(* IEC 61131-3 sources: eCockpitGit/test_project/src/%F%00 Library/%F%Common Functions/%F%Bits/%F%Bit Get, 3 files *)

(* ---- %POU%FU_bBitGet.st ---- *)
//This function get the bit value from a variable
// |**Version**|**Author**| **Date** |**Changes**
// | 1         | NSN      | 11-01-19 | Creation
FUNCTION FU_bBitGet : BOOL
VAR_INPUT
	bVar	:BYTE;		//The value to work with
	bIndex	:BYTE;		//Which bit to get
END_VAR
(*%!%__DELIMITER__%!%*)
FU_bBitGet			:=		(bVar AND SHL(1,bIndex)) <> 0;

(* ---- %POU%FU_dwBitGet.st ---- *)
//This function get the bit value from a variable
// |**Version**|**Author**| **Date** |**Changes**
// | 1         | NSN      | 11-01-19 | Creation
FUNCTION FU_dwBitGet : BOOL
VAR_INPUT
	dbVar	:DWORD;		//The value to work with
	bIndex	:BYTE;		//Which bit to get
END_VAR
(*%!%__DELIMITER__%!%*)
FU_dwBitGet		:=		(dbVar AND SHL(1,bIndex)) <> 0;

(* ---- %POU%FU_wBitGet.st ---- *)
//This function get the bit value from a variable
// |**Version**|**Author**| **Date** |**Changes**
// | 1         | NSN      | 11-01-19 | Creation
FUNCTION FU_wBitGet : BOOL
VAR_INPUT
	wVar	:WORD;		//The value to work with
	bIndex	:BYTE;		//Which bit to get
END_VAR
(*%!%__DELIMITER__%!%*)
FU_wBitGet		:=		(wVar AND SHL(1,bIndex)) <> 0;
